(*
Nazwa:			E_LidFeederState
Opis:			Stan zpodajnika platynek
Wersja:			v0.2
Data:			2018-10-18
Autor:			TW
Urzadzenia:		
Konfiguracja:	
Info:
*)

TYPE E_WickFeederState :
(
	eDisabled:=0,	//Wyłączona
	eError:=1,		//Błąd
	eManualMovement:=2,	//Tryb serwisowy
	eHoming:=3,		//Bazowanie
	eHomingDone:=4,	//Koniec bazowania
	//eHeaterNotReady:=5,	//Grzanie
	eFilling:=5,  //Zapełnianie zasobników
	eReady:=6,		//Gotowość 
	eWickDepotReady:=7,	//Magazynek przed włożeniem
	ePuttingWick:=8,	//Przygotowanie do odlożenia
	//ePuttingLid2:=9,	//Nakładanie ostatnie
	//eHeating:=10,	//Zgrzewanie
	eWickPutted:=11,	//Odłożona
	eGoingUp:=12,	//Podnoszenie
	ePreparingToDisable:=13 (*NOWY*) //Przygotowanie do wyłączenia
(**)
):=eDisabled;
END_TYPE

(* stored: Version 1.2.0.0, ProductVersion 3.1.4026.13, FileIdentifier b4677336a0cbf3a481fa803b6cc691517af9174b, FileSignature 628968bce00b5535e68312c159fa9833896ad82965d99abd1c8637b7ddc456f55900d0cb0026d56ab2c19467bcbd3596a0739ea41f586e64e6ef1d5002929d723bb04eb2d866a29a28f172faf254df21773a2e7dd756b043cc533c4b4da6007f12ddc470bb5a46adcbbf3d515b653665077c47a18fb4e3b73ad5ae9717216e665a08e90f80fcc138117b0d350009425826704a59cdd5cd394d3a7b7d39b0e886037624fccd54823c9b3e0c603d86542df994795221bc66d5affdaf0c13d8d9dd121a51be7db8d0c0a932e207fe2bb8e48b9591e72d9d1c33164901bbaaa2bde0b8cb6f7d485fe650a7c29e8f66ed2c95036b302984184ba8ae0c44ea0989fa51
   DUT E_WickFeederState: Id {6a4536bb-da18-4cdd-9ce8-1808bd978415} *)
